TYPE E_Command :
(
    none := 0,
    Start,
    Stop,
	MoveSlaveVelo,
    Reset
);
END_TYPE

(* stored: Version 1.1.0.1
   DUT E_Command: Id {572bd783-d8fe-401a-8175-95194f46609a} *)
